// TIA Portal V18 export
// export: Created 2025-12-01T17:53:10.2052164Z, ExportSetting None, DisplayName Totally Integrated Automation Portal, DisplayVersion V18 Update 5, DisplayName TIA Portal Openness, DisplayVersion V18 Update 5, DisplayName TIA Portal Teamcenter Gateway, DisplayVersion V18, DisplayName TIA Portal Version Control Interface, DisplayVersion V18, DisplayName STEP 7 Professional, DisplayVersion V18 Update 5, DisplayName STEP 7 Safety, DisplayVersion V18, DisplayName WinCC Professional, DisplayVersion V18 Update 5
Screen "617DP_Frame"  1280x800, Number=617, Template=06Diagnosis
  ScreenLayer 
    GraphicView "图形视图_1" at 5,98 size 1266x578  Picture=图形_21
